TYPE T_RejectCode : STRING[100];
END_TYPE

(* stored: Version 1.1.0.1, ProductVersion 3.1.4024.15
   DUT T_RejectCode: Id {7805a772-8364-4085-a35d-dce6c88b65b6} *)
